FUNCTION_BLOCK FB_MachineState
VAR_INPUT
	bBase				:BOOL :=TRUE;		//何もなし
	bCritical			:BOOL;				//クリティカルの発生
	bError				:BOOL;				//エラーの発生
	bWarning			:BOOL;				//ワーニングの発生
	bStay				:BOOL;				//McPowerがOFF
	bStop				:BOOL;				//McPowerがON
	bMoving				:BOOL;				//軸動作中

END_VAR
VAR_OUTPUT
	eMachineState		:E_MachineState;	//マシーンステートを出力
	bStopMachine		:BOOL;				//モーションファンクションブロック停止
END_VAR
VAR
	i					:INT:=1;
	al_index			:INT:=1;
	p_alarms			: ARRAY [1..GVL_Alarm.iMaxAlarm] OF POINTER TO FB_Alarm;
END_VAR

//--発生中アラームを集計---
	//アラームをリセット
	THIS^.bCritical:=FALSE;
	THIS^.bError:=FALSE;
	THIS^.bError:=FALSE;
	
	//アラーム集計
	FOR i := 1	TO al_index -1  BY 1 DO
		CASE p_alarms[i]^.eSeverity OF
			TcEventSeverity.Critical:
				IF p_alarms[i]^.bRaised=TRUE THEN
					THIS^.bCritical:=TRUE;
				END_IF
				
			TcEventSeverity.Error:
				IF p_alarms[i]^.bRaised=TRUE THEN
					THIS^.bError:=TRUE;
				END_IF
			
			TcEventSeverity.Warning:
				IF p_alarms[i]^.bRaised=TRUE THEN
					THIS^.bWarning:=TRUE;
				END_IF
			
		END_CASE
		
	END_FOR


//---発生アラームの重いほうからマシンステートに登録---
	IF bCritical=TRUE THEN
		eMachineState:=E_MachineState.Critical;
		bStopMachine:=TRUE;
		
	ELSIF bError=TRUE THEN
		eMachineState:=E_MachineState.Error;
		bStopMachine:=TRUE;
	
	ELSIF bWarning=TRUE THEN
		eMachineState:=E_MachineState.Warning;
		bStopMachine:=FALSE;
		
	ELSIF bStay=TRUE THEN
		eMachineState:=E_MachineState.Stay;
		bStopMachine:=FALSE;
		
	ELSIF bStop=TRUE THEN
		eMachineState:=E_MachineState.Stop;
		bStopMachine:=FALSE;
		
	ELSIF bMoving=TRUE THEN
		eMachineState:=E_MachineState.Moving;
		bStopMachine:=FALSE;

	ELSIF bBase=TRUE THEN
		eMachineState:=E_MachineState.Base;
		bStopMachine:=FALSE;
	END_IF

METHOD reg_alarm : BOOL
VAR_INPUT
	p_alarm	:POINTER TO FB_Alarm;
END_VAR
IF GVL_Alarm.iMaxAlarm < al_index THEN
	reg_alarm:=FALSE;
	RETURN;
END_IF

p_alarms[al_index] := p_alarm;
al_index := al_index + 1;
reg_alarm:=TRUE;
END_METHOD

END_FUNCTION_BLOCK

(* stored: Version 1.1.0.1, ProductVersion 3.1.4024.12
   POU FB_MachineState: Id {c973bc40-a96e-4db3-9daa-2f59595f3f57}, SpecialFunc None
   Method reg_alarm: Id {c7217401-5976-4e6a-8be4-b75e078b5d2f} *)
